(* Logix 5000 project; controller StartingFile_Isaiah_Regacho vendor 1 type 14 code 106 rev 28.11; software revision 28.03 *)

TASK Fault_Logging (periodic, rate 100 ms, priority 10, watchdog 500 ms) : Fault_Logging_Program   // Logs data on faults
TASK MainTask (continuous, watchdog 500 ms) : MainProgram

MODULES
   Local : vendor 1 type 14 code 106 (Compact 0, rev 28.11)
       : 1769-IQ16 (Compact 3, rev 1.1, Input RPI 20 ms)
       : vendor 1 type 7 code 77 (Compact 2, rev 3.1, Input RPI 20 ms)
       : vendor 1 type 7 code 72 (Compact 4, rev 2.1, Output RPI 20 ms)
       : vendor 1 type 7 code 72 (Compact 5, rev 2.1, Output RPI 20 ms)
END_MODULES

TYPE DATE_TIME :
STRUCT
   dateTime : DINT[7];
END_STRUCT
END_TYPE

TYPE FAULTS :
STRUCT
   faultCode : DINT;   // custom fault code depending on type of fault
   timeFaulted : DINT[7];   // time the fault occured
   faultType : DINT;   // minor (1) or major (2) fault
   systemState : DINT;   // current elevator floor state when the fault occured
END_STRUCT
END_TYPE

TYPE LOG_DATA :
STRUCT
   numCalls : DINT;   // keeps track of the # of calls a floor made. also is used for indexing the serviceLog
   timeAve : DINT;   // the average time it takes to service floor
   serviceLog : DATE_TIME[50];   // log of all times a floor was serviced
   timeAcc : DINT;   // keeps track of the TOTAL service time. must divide by numCalls to find average
   timeService : DINT;   // the time it takes to service a floor one instance
END_STRUCT
END_TYPE

ADD_ON_INSTRUCTION getFloorData   (* revision 1.0, ExecutePrescan, ExecuteEnableInFalse *)
// gets floor data and stores in masterLog
VAR_IN_OUT
   floorLogData : LOG_DATA; {required}
END_VAR
VAR
   timeCount : TIMER; {access None}
   logIndex : DINT; {access None}
   false_ons : BOOL; {access None}
END_VAR

ROUTINE EnableInFalse   (* ladder *)
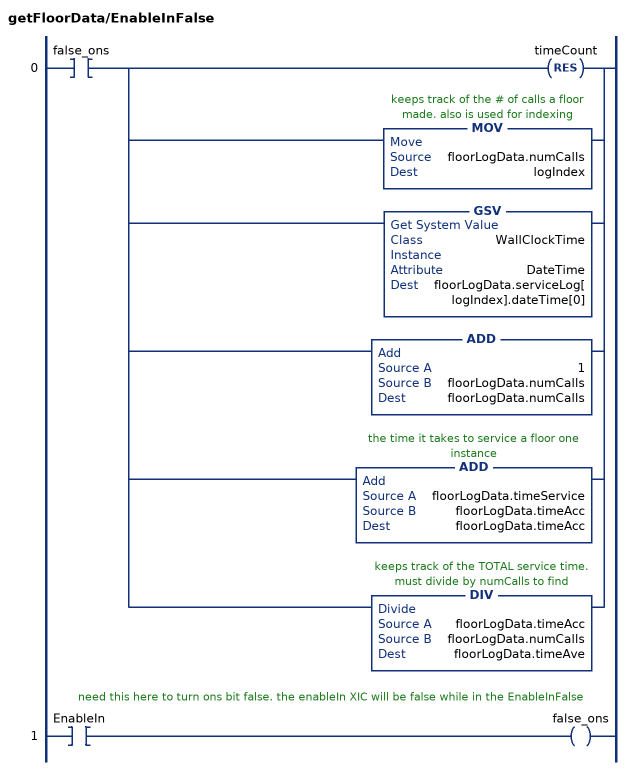
   0: XIC(false_ons)[RES(timeCount) ,MOV(floorLogData.numCalls,logIndex) ,GSV(WallClockTime,,DateTime,floorLogData.serviceLog[logIndex].dateTime[0]) ,ADD(1,floorLogData.numCalls,floorLogData.numCalls) ,ADD(floorLogData.timeService,floorLogData.timeAcc,floorLogData.timeAcc) ,DIV(floorLogData.timeAcc,floorLogData.numCalls,floorLogData.timeAve) ];
   // need this here to turn ons bit false. the enableIn XIC will be false while in the EnableInFalse
   1: XIC(EnableIn)OTE(false_ons);
END_ROUTINE

ROUTINE Logic   (* ladder *)
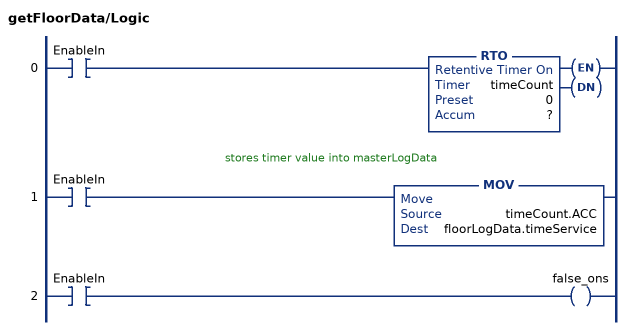
   0: XIC(EnableIn)RTO(timeCount,?,?);
   // stores timer value into masterLogData
   1: XIC(EnableIn)MOV(timeCount.ACC,floorLogData.timeService);
   2: XIC(EnableIn)OTE(false_ons);
END_ROUTINE

ROUTINE Prescan   (* ladder *)
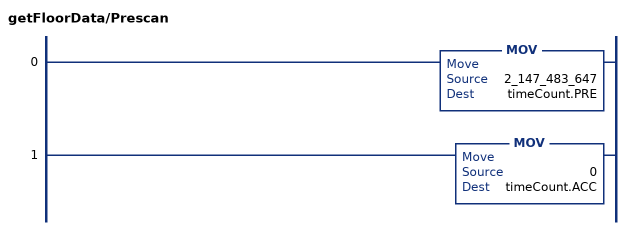
   0: MOV(2_147_483_647,timeCount.PRE);
   1: MOV(0,timeCount.ACC);
END_ROUTINE
END_ADD_ON_INSTRUCTION

PROGRAM Fault_Logging_Program   (* main routine Fault_Logging_Routine *)
VAR
   doorOpenFault_ons : BOOL;
   doorOpenFaultBit : BOOL;
   index : DINT;
   masterFaultLog : FAULTS[10];
   motorRunFault_ons : BOOL;
   motorRunFaultBit : BOOL;
   sensorFault_ons : BOOL;
   sensorFaultBit : BOOL;
END_VAR

ROUTINE Fault_Logging_Routine   (* ladder *)
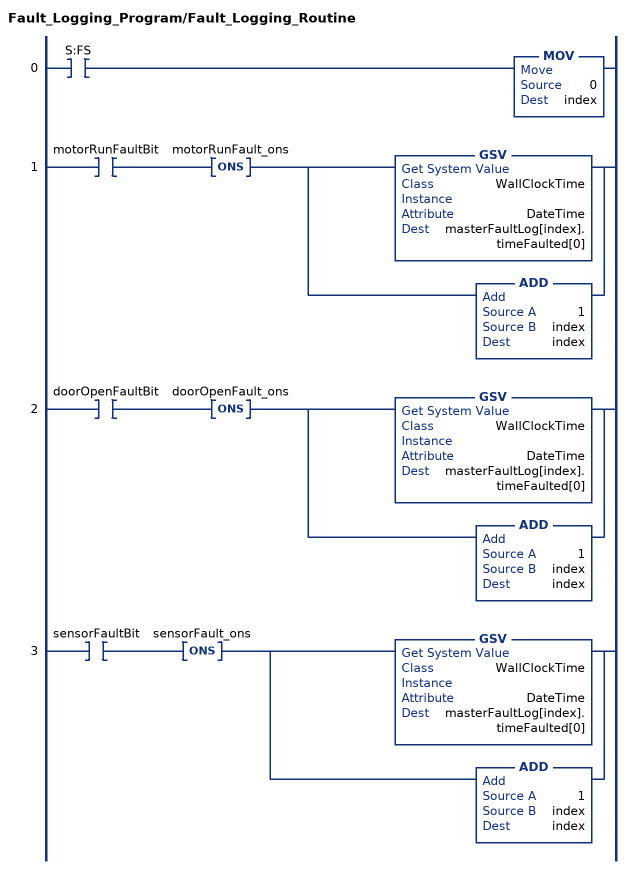
   0: XIC(S:FS)MOV(0,index);
   1: XIC(motorRunFaultBit)ONS(motorRunFault_ons)[GSV(WallClockTime,,DateTime,masterFaultLog[index].timeFaulted[0]) ,ADD(1,index,index) ];
   2: XIC(doorOpenFaultBit)ONS(doorOpenFault_ons)[GSV(WallClockTime,,DateTime,masterFaultLog[index].timeFaulted[0]) ,ADD(1,index,index) ];
   3: XIC(sensorFaultBit)ONS(sensorFault_ons)[GSV(WallClockTime,,DateTime,masterFaultLog[index].timeFaulted[0]) ,ADD(1,index,index) ];
END_ROUTINE
END_PROGRAM

PROGRAM MainProgram   (* main routine MainRoutine *)
VAR
   breakpoint_ons : BOOL;
   callArray : DINT[6] := ([1] := 1, [2] := 2, [4] := 4);
   checkedBothDir : DINT;
   clearFaultsBit : BOOL;
   control_1 : CONTROL := (LEN := 4, EN := 1, IN := 1, FD := 1);
   countDown_ons : BOOL;
   countUp_ons : BOOL;
   CR0 : ALIAS FOR Local:5:O.Data.4;   // Control Relay 0
   Current_State : DINT := 100;
   Current_State_Door : DINT := 1;
   currentFloor : DINT := 4;
   DCLS : ALIAS FOR Local:3:I.Data.8;   // Door Close Limit Switch
   DOLS : ALIAS FOR Local:3:I.Data.9;   // Door Open Limit Switch
   doorOpenFault : TIMER := (PRE := 10000);
   doorOpenFault_ons : BOOL;
   doorOpenFaultBit : BOOL;
   doorOpenFunc : DINT;
   down_ons : BOOL;
   elevatorDirection : DINT;
   faultIndex : DINT;
   FIL1 : ALIAS FOR Local:4:O.Data.11;   // Floor Indicator Light 1
   FIL2 : ALIAS FOR Local:4:O.Data.10;   // Floor Indicator Light 2
   FIL3 : ALIAS FOR Local:4:O.Data.9;   // Floor Indicator Light 3
   FIL4 : ALIAS FOR Local:4:O.Data.8;   // Floor Indicator Light 4
   floor1 : DINT;
   floor1_ons : BOOL;
   floor1Data : getFloorData;
   floor2 : DINT := 1;
   floor2_ons : BOOL;
   floor2Data : getFloorData;
   floor3 : DINT := 2;
   floor3_ons : BOOL;
   floor3Data : getFloorData;
   floor4 : DINT := 3;
   floor4_ons : BOOL;
   floor4Data : getFloorData;
   FLS1 : ALIAS FOR Local:3:I.Data.0;   // Floor Limit Switch 1
   FLS2 : ALIAS FOR Local:3:I.Data.1;   // Floor Limit Switch 2
   FLS3 : ALIAS FOR Local:3:I.Data.2;   // Floor Limit Switch 3
   FLS4 : ALIAS FOR Local:3:I.Data.3;   // Floor Limit Switch 4
   FPB1 : ALIAS FOR Local:2:I.Data.11;   // Floor Pushbutton 1
   FPB2 : ALIAS FOR Local:2:I.Data.10;   // Floor Pushbutton 2
   FPB3 : ALIAS FOR Local:2:I.Data.9;   // Floor Pushbutton 3
   FPB4 : ALIAS FOR Local:2:I.Data.8;   // Floor Pushbutton 4
   IL1 : ALIAS FOR Local:4:O.Data.3;   // Indicator Light 1
   IL2 : ALIAS FOR Local:4:O.Data.2;   // Indicator Light 2
   IL3 : ALIAS FOR Local:4:O.Data.1;   // Indicator Light 3
   IL4 : ALIAS FOR Local:4:O.Data.0;   // Indicator Light 4
   ILC : ALIAS FOR Local:4:O.Data.5;   // Indicator Light Close
   ILE5 : ALIAS FOR Local:4:O.Data.6;   // Indicator Light Emergency 5
   ILO : ALIAS FOR Local:4:O.Data.4;   // Indicator Light Open
   ILTS0 : ALIAS FOR Local:4:O.Data.14;   // Indicator Light Toggle Switch 0
   ILTS1 : ALIAS FOR Local:4:O.Data.13;   // Indicator Light Toggle Switch 1
   ILTS2 : ALIAS FOR Local:4:O.Data.12;   // Indicator Light Toggle Switch 2
   index : DINT := 5;
   logIndex : DINT;
   M0 : ALIAS FOR Local:5:O.Data.0;   // Motor 0
   majorFault_var : DINT := 1;
   masterFaultLog : FAULTS[10];
   masterFaultLog_init : FAULTS[10];
   masterLogData : LOG_DATA[4] := ([0].numCalls := 3, [0].timeAve := 6729, [0].serviceLog[0].dateTime[0] := 2024, [0].serviceLog[0].dateTime[1] := 4, [0].serviceLog[0].dateTime[2] := 11, [0].serviceLog[0].dateTime[3] := 12, [0].serviceLog[0].dateTime[4] := 6, [0].serviceLog[0].dateTime[5] := 16, [0].serviceLog[0].dateTime[6] := 127621, [0].serviceLog[1].dateTime[0] := 2024, [0].serviceLog[1].dateTime[1] := 4, [0].serviceLog[1].dateTime[2] := 11, [0].serviceLog[1].dateTime[3] := 12, [0].serviceLog[1].dateTime[4] := 6, [0].serviceLog[1].dateTime[5] := 34, [0].serviceLog[1].dateTime[6] := 745369, [0].serviceLog[2].dateTime[0] := 2024, [0].serviceLog[2].dateTime[1] := 4, [0].serviceLog[2].dateTime[2] := 11, [0].serviceLog[2].dateTime[3] := 12, [0].serviceLog[2].dateTime[4] := 7, [0].serviceLog[2].dateTime[5] := 4, [0].serviceLog[2].dateTime[6] := 869689, [0].timeAcc := 20188, [0].timeService := 363313, [1].numCalls := 2, [1].timeAve := 12433, [1].serviceLog[0].dateTime[0] := 2024, [1].serviceLog[0].dateTime[1] := 4, [1].serviceLog[0].dateTime[2] := 11, [1].serviceLog[0].dateTime[3] := 12, [1].serviceLog[0].dateTime[4] := 6, [1].serviceLog[0].dateTime[5] := 10, [1].serviceLog[0].dateTime[6] := 288799, [1].serviceLog[1].dateTime[0] := 2024, [1].serviceLog[1].dateTime[1] := 4, [1].serviceLog[1].dateTime[2] := 11, [1].serviceLog[1].dateTime[3] := 12, [1].serviceLog[1].dateTime[4] := 6, [1].serviceLog[1].dateTime[5] := 45, [1].serviceLog[1].dateTime[6] := 652417, [1].timeAcc := 24866, [1].timeService := 363928, [3].numCalls := 4, [3].timeAve := 8386, [3].serviceLog[0].dateTime[0] := 2024, [3].serviceLog[0].dateTime[1] := 4, [3].serviceLog[0].dateTime[2] := 11, [3].serviceLog[0].dateTime[3] := 12, [3].serviceLog[0].dateTime[4] := 6, [3].serviceLog[0].dateTime[5] := 3, [3].serviceLog[0].dateTime[6] := 427814, [3].serviceLog[1].dateTime[0] := 2024, [3].serviceLog[1].dateTime[1] := 4, [3].serviceLog[1].dateTime[2] := 11, [3].serviceLog[1].dateTime[3] := 12, [3].serviceLog[1].dateTime[4] := 6, [3].serviceLog[1].dateTime[5] := 22, [3].serviceLog[1].dateTime[6] := 780797, [3].serviceLog[2].dateTime[0] := 2024,
        [3].serviceLog[2].dateTime[1] := 4, [3].serviceLog[2].dateTime[2] := 11, [3].serviceLog[2].dateTime[3] := 12, [3].serviceLog[2].dateTime[4] := 6, [3].serviceLog[2].dateTime[5] := 49, [3].serviceLog[2].dateTime[6] := 470088, [3].serviceLog[3].dateTime[0] := 2024, [3].serviceLog[3].dateTime[1] := 4, [3].serviceLog[3].dateTime[2] := 11, [3].serviceLog[3].dateTime[3] := 12, [3].serviceLog[3].dateTime[4] := 6, [3].serviceLog[3].dateTime[5] := 56, [3].serviceLog[3].dateTime[6] := 856063, [3].timeAcc := 33544, [3].timeService := 364724);
   masterLogData_init : LOG_DATA[4];
   motorRunFault : TIMER := (PRE := 8000);
   motorRunFault_ons : BOOL;
   motorRunFaultBit : BOOL;
   Next_State : DINT := 100;
   Next_State_Door : DINT := 1;
   nextFloor : DINT := 4;
   PB1 : ALIAS FOR Local:2:I.Data.3;   // Pushbutton 1
   PB2 : ALIAS FOR Local:2:I.Data.2;   // Pushbutton 2
   PB3 : ALIAS FOR Local:2:I.Data.1;   // Pushbutton 3
   PB4 : ALIAS FOR Local:2:I.Data.0;   // Pushbutton 4
   PBC : ALIAS FOR Local:2:I.Data.5;   // Pushbutton Close
   PBE5 : ALIAS FOR Local:2:I.Data.6;   // Pushbutton Emergency 5
   PBO : ALIAS FOR Local:2:I.Data.4;   // Pushbutton Open
   sensorFault_ons : BOOL;
   sensorFaultBit : BOOL;
   SOL0 : ALIAS FOR Local:5:O.Data.2;   // Solenoid 0
   START : ALIAS FOR Local:2:I.Data.14;   // Start Button (N.O.)
   STOP : ALIAS FOR Local:2:I.Data.15;   // Stop Button (N.C.)
   test2_ons : BOOL;
   test_ons : BOOL;
   timer3sec : TIMER := (PRE := 3000, ACC := 3000, EN := 1, DN := 1);
   timer3secVar : DINT := 1;
   timer5sec : TIMER := (PRE := 5000, ACC := 5000, EN := 1, DN := 1);
   TS0 : ALIAS FOR Local:3:I.Data.12;   // Toggle Switch 0
   TS1 : ALIAS FOR Local:3:I.Data.11;   // Toggle Switch 1
   TS2 : ALIAS FOR Local:3:I.Data.10;   // Toggle Switch 2
   up_ons : BOOL;
   V_CR0 : BOOL;   // Virtual Control Relay 0
   V_DCLS : BOOL;   // Virtual Door Close Limit Switch
   V_DOLS : BOOL := 1;   // Virtual Door Open Limit Switch
   V_FIL1 : BOOL := 1;   // Virtual Floor Indicator Light 1
   V_FIL2 : BOOL := 1;   // Virtual Floor Indicator Light 2
   V_FIL3 : BOOL;   // Virtual Floor Indicator Light 3
   V_FIL4 : BOOL := 1;   // Virtual Floor Indicator Light 4
   V_FLS1 : BOOL;   // Virtual Floor Limit Switch 1
   V_FLS2 : BOOL;   // Virtual Floor Limit Switch 2
   V_FLS3 : BOOL;   // Virtual Floor Limit Switch 3
   V_FLS4 : BOOL;   // Virtual Floor Limit Switch 4
   V_FPB1 : BOOL;   // Virtual Floor Pushbutton 1
   V_FPB2 : BOOL;   // Virtual Floor Pushbutton 2
   V_FPB3 : BOOL;   // Virtual Floor Pushbutton 3
   V_FPB4 : BOOL;   // Virtual Floor Pushbutton 4
   V_IL1 : BOOL := 1;   // Virtual Indicator Light 1
   V_IL2 : BOOL := 1;   // Virtual Indicator Light 2
   V_IL3 : BOOL;   // Virtual Indicator Light 3
   V_IL4 : BOOL := 1;   // Virtual Indicator Light 4
   V_ILC : BOOL := 1;   // Virtual Indicator Light Close
   V_ILE5 : BOOL := 1;   // Virtual Indicator Light Emergency 5
   V_ILO : BOOL;   // Virtual Indicator Light Open
   V_ILTS0 : BOOL;   // Vitual Indicator Light Toggle Switch 0
   V_ILTS1 : BOOL;   // Virtual Indicator Light Toggle Switch 1
   V_ILTS2 : BOOL;   // Virtual Indicator Light Toggle Switch 2
   V_M0 : BOOL;   // Virtual Motor 0
   V_PB1 : BOOL;   // Virtual Pushbutton 1
   V_PB2 : BOOL;   // Virtual Pushbutton 2
   V_PB3 : BOOL;   // Virtual Pushbutton 3
   V_PB4 : BOOL;   // Virtual Pushbutton 4
   V_PBC : BOOL;   // Virtual Pushbutton Close
   V_PBE5 : BOOL;   // Virtual Pushbutton Emergency 5
   V_PBO : BOOL;   // Virtual Pushbutton Open
   V_SOL0 : BOOL := 1;   // Virtual Solenoid 0
   V_START : BOOL;   // Virtual Start Button (N.O.)
   V_STOP : BOOL := 1;   // Virtual Stop Button (N.C.)
   V_TS0 : BOOL := 1;   // Virtual Toggle Switch 0
   V_TS1 : BOOL;   // Virtual Toggle Switch 1
   V_TS2 : BOOL;   // Virtual Toggle Switch 2
END_VAR

ROUTINE BufferInput   (* ladder *)
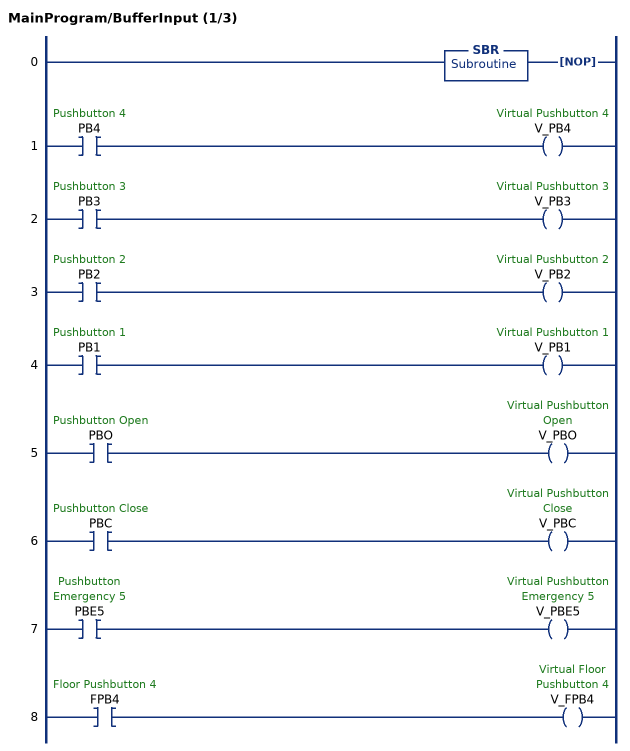
   0: SBR()NOP();
   1: XIC(PB4)OTE(V_PB4);
   2: XIC(PB3)OTE(V_PB3);
   3: XIC(PB2)OTE(V_PB2);
   4: XIC(PB1)OTE(V_PB1);
   5: XIC(PBO)OTE(V_PBO);
   6: XIC(PBC)OTE(V_PBC);
   7: XIC(PBE5)OTE(V_PBE5);
   8: XIC(FPB4)OTE(V_FPB4);
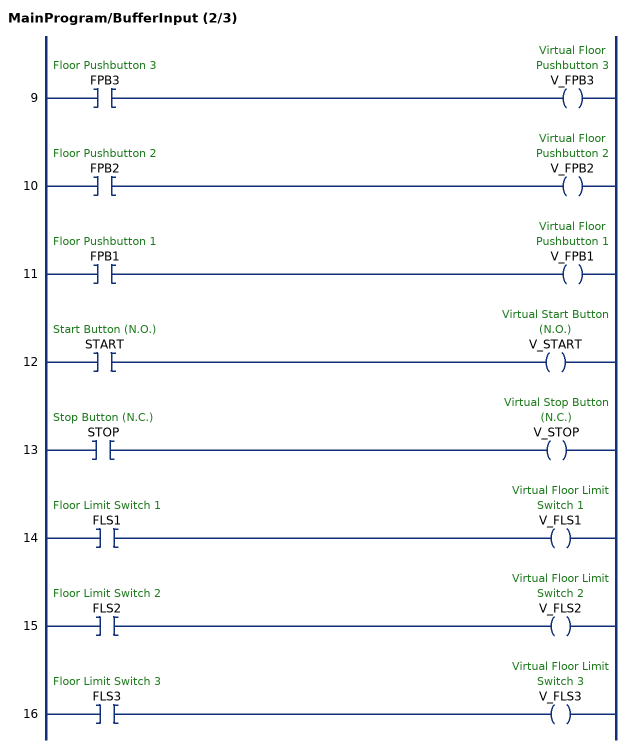
   9: XIC(FPB3)OTE(V_FPB3);
   10: XIC(FPB2)OTE(V_FPB2);
   11: XIC(FPB1)OTE(V_FPB1);
   12: XIC(START)OTE(V_START);
   13: XIC(STOP)OTE(V_STOP);
   14: XIC(FLS1)OTE(V_FLS1);
   15: XIC(FLS2)OTE(V_FLS2);
   16: XIC(FLS3)OTE(V_FLS3);
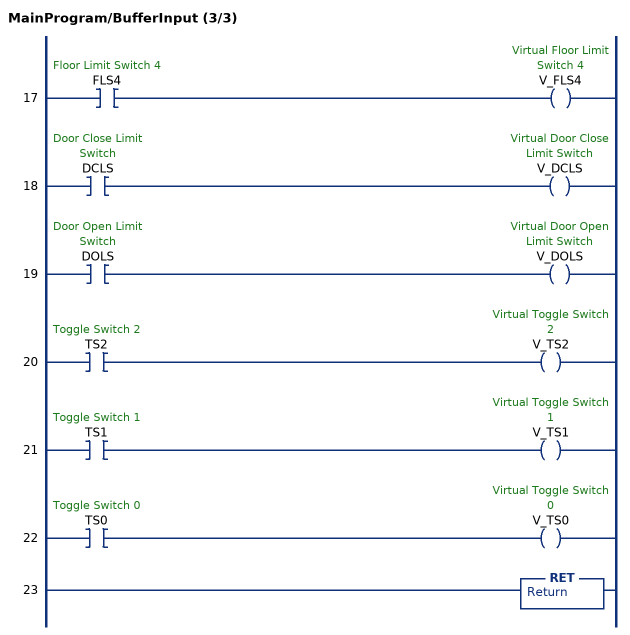
   17: XIC(FLS4)OTE(V_FLS4);
   18: XIC(DCLS)OTE(V_DCLS);
   19: XIC(DOLS)OTE(V_DOLS);
   20: XIC(TS2)OTE(V_TS2);
   21: XIC(TS1)OTE(V_TS1);
   22: XIC(TS0)OTE(V_TS0);
   23: RET();
END_ROUTINE

ROUTINE BufferOutput   (* ladder *)
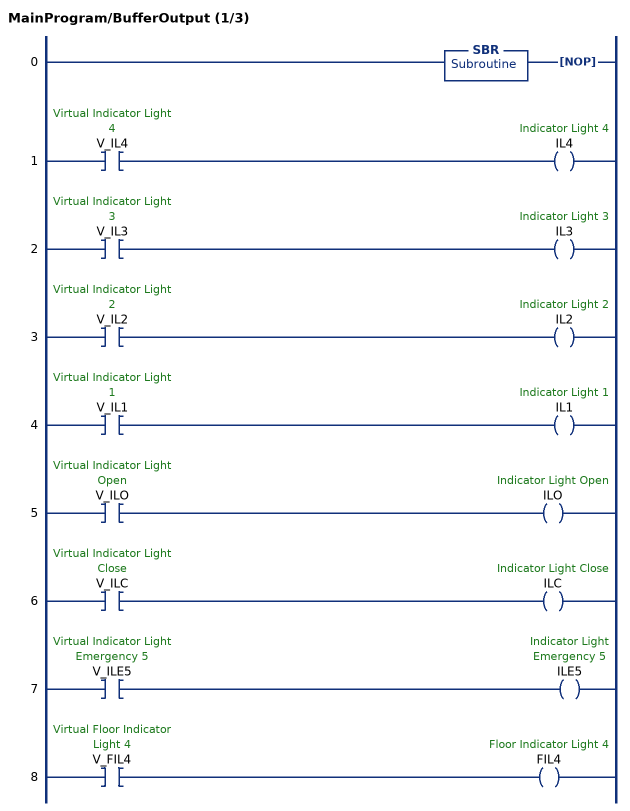
   0: SBR()NOP();
   1: XIC(V_IL4)OTE(IL4);
   2: XIC(V_IL3)OTE(IL3);
   3: XIC(V_IL2)OTE(IL2);
   4: XIC(V_IL1)OTE(IL1);
   5: XIC(V_ILO)OTE(ILO);
   6: XIC(V_ILC)OTE(ILC);
   7: XIC(V_ILE5)OTE(ILE5);
   8: XIC(V_FIL4)OTE(FIL4);
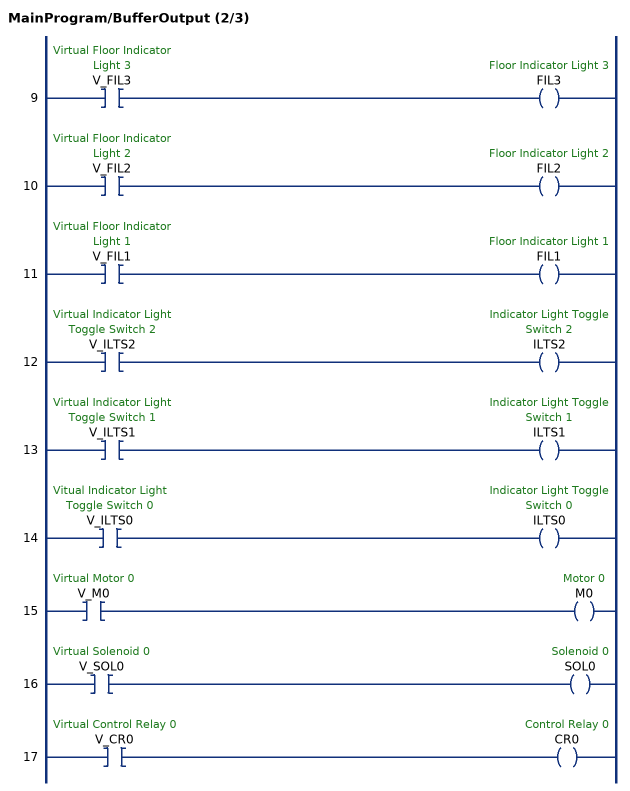
   9: XIC(V_FIL3)OTE(FIL3);
   10: XIC(V_FIL2)OTE(FIL2);
   11: XIC(V_FIL1)OTE(FIL1);
   12: XIC(V_ILTS2)OTE(ILTS2);
   13: XIC(V_ILTS1)OTE(ILTS1);
   14: XIC(V_ILTS0)OTE(ILTS0);
   15: XIC(V_M0)OTE(M0);
   16: XIC(V_SOL0)OTE(SOL0);
   17: XIC(V_CR0)OTE(CR0);
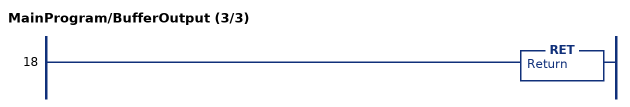
   18: RET();
END_ROUTINE

ROUTINE Door_State_Machine   (* ladder *)
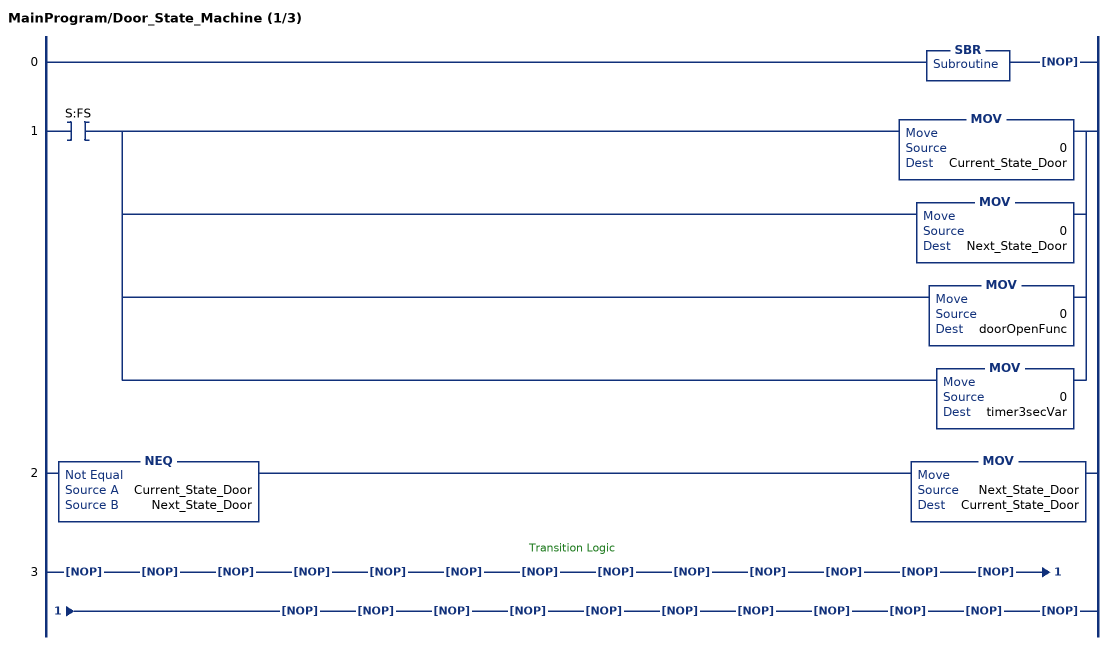
   0: SBR()NOP();
   1: XIC(S:FS)[MOV(0,Current_State_Door) ,MOV(0,Next_State_Door) ,MOV(0,doorOpenFunc) ,MOV(0,timer3secVar) ];
   2: NEQ(Current_State_Door,Next_State_Door)MOV(Next_State_Door,Current_State_Door);
   // Transition Logic
   3: NOP()NOP()NOP()NOP()NOP()NOP()NOP()NOP()NOP()NOP()NOP()NOP()NOP()NOP()NOP()NOP()NOP()NOP()NOP()NOP()NOP()NOP()NOP()NOP();
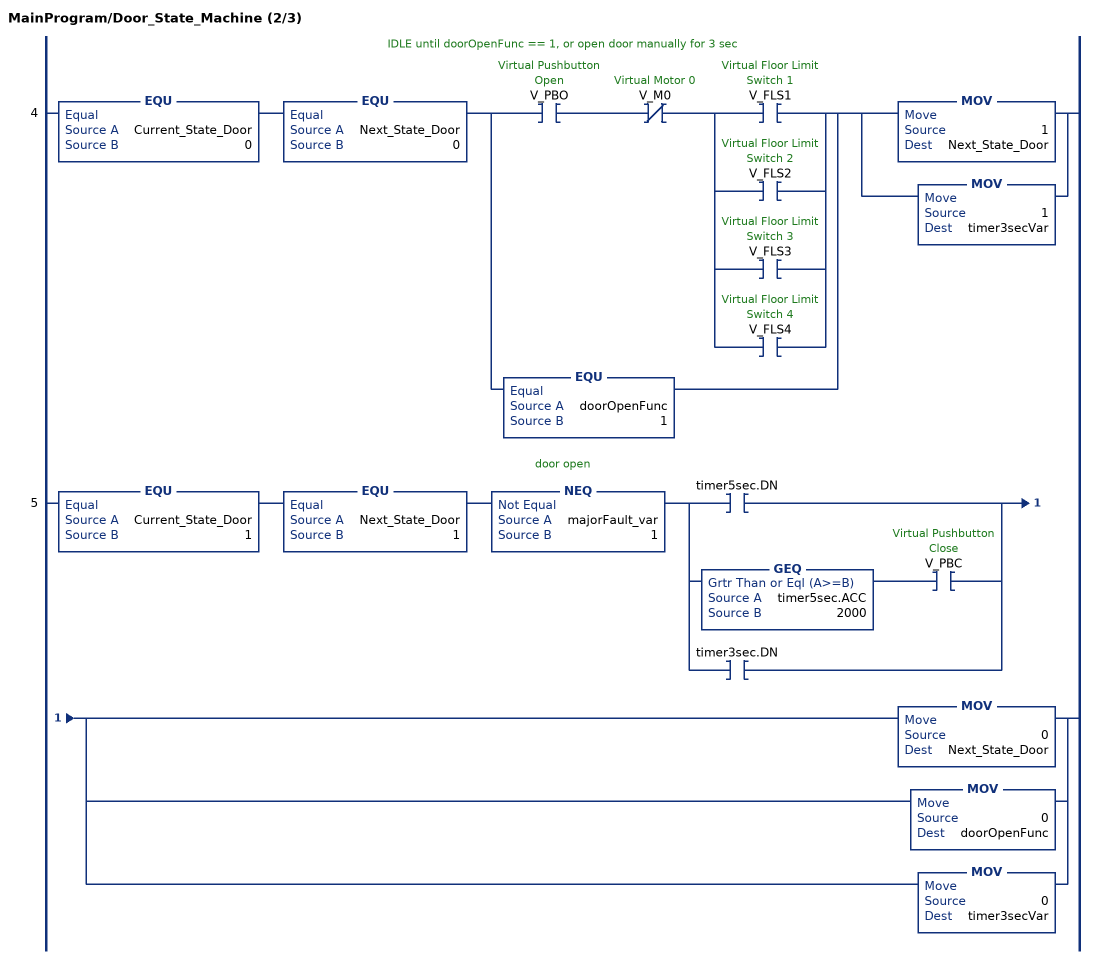
   // IDLE until doorOpenFunc == 1, or open door manually for 3 sec
   4: EQU(Current_State_Door,0)EQU(Next_State_Door,0)[XIC(V_PBO) XIO(V_M0) [XIC(V_FLS1) ,XIC(V_FLS2) ,XIC(V_FLS3) ,XIC(V_FLS4) ] ,EQU(doorOpenFunc,1) ][MOV(1,Next_State_Door) ,MOV(1,timer3secVar) ];
   // door open
   5: EQU(Current_State_Door,1)EQU(Next_State_Door,1)NEQ(majorFault_var,1)[XIC(timer5sec.DN) ,GEQ(timer5sec.ACC,2000) XIC(V_PBC) ,XIC(timer3sec.DN) ][MOV(0,Next_State_Door) ,MOV(0,doorOpenFunc) ,MOV(0,timer3secVar) ];
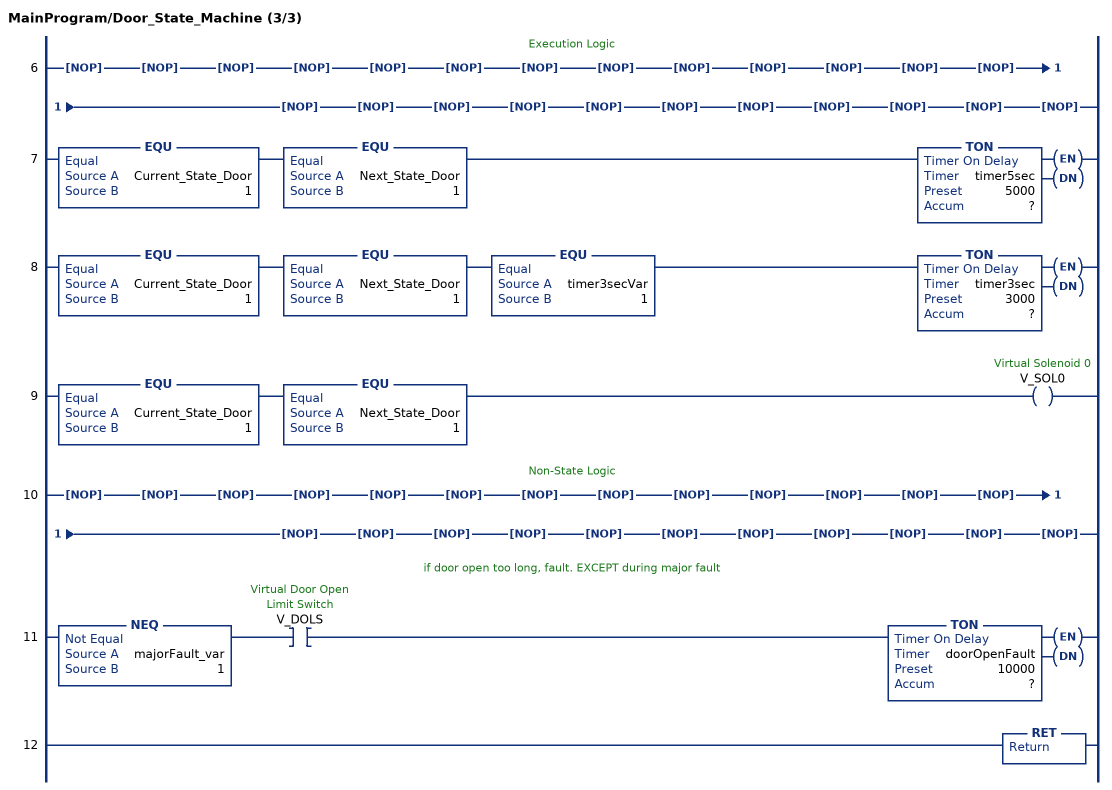
   // Execution Logic
   6: NOP()NOP()NOP()NOP()NOP()NOP()NOP()NOP()NOP()NOP()NOP()NOP()NOP()NOP()NOP()NOP()NOP()NOP()NOP()NOP()NOP()NOP()NOP()NOP();
   7: EQU(Current_State_Door,1)EQU(Next_State_Door,1)TON(timer5sec,?,?);
   8: EQU(Current_State_Door,1)EQU(Next_State_Door,1)EQU(timer3secVar,1)TON(timer3sec,?,?);
   9: EQU(Current_State_Door,1)EQU(Next_State_Door,1)OTE(V_SOL0);
   // Non-State Logic
   10: NOP()NOP()NOP()NOP()NOP()NOP()NOP()NOP()NOP()NOP()NOP()NOP()NOP()NOP()NOP()NOP()NOP()NOP()NOP()NOP()NOP()NOP()NOP()NOP();
   // if door open too long, fault. EXCEPT during major fault
   11: NEQ(majorFault_var,1)XIC(V_DOLS)TON(doorOpenFault,?,?);
   12: RET();
END_ROUTINE

ROUTINE Floor_State_Machine   (* ladder *)
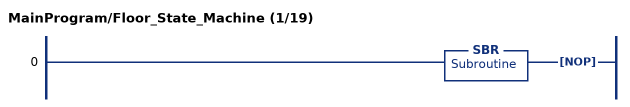
   0: SBR()NOP();
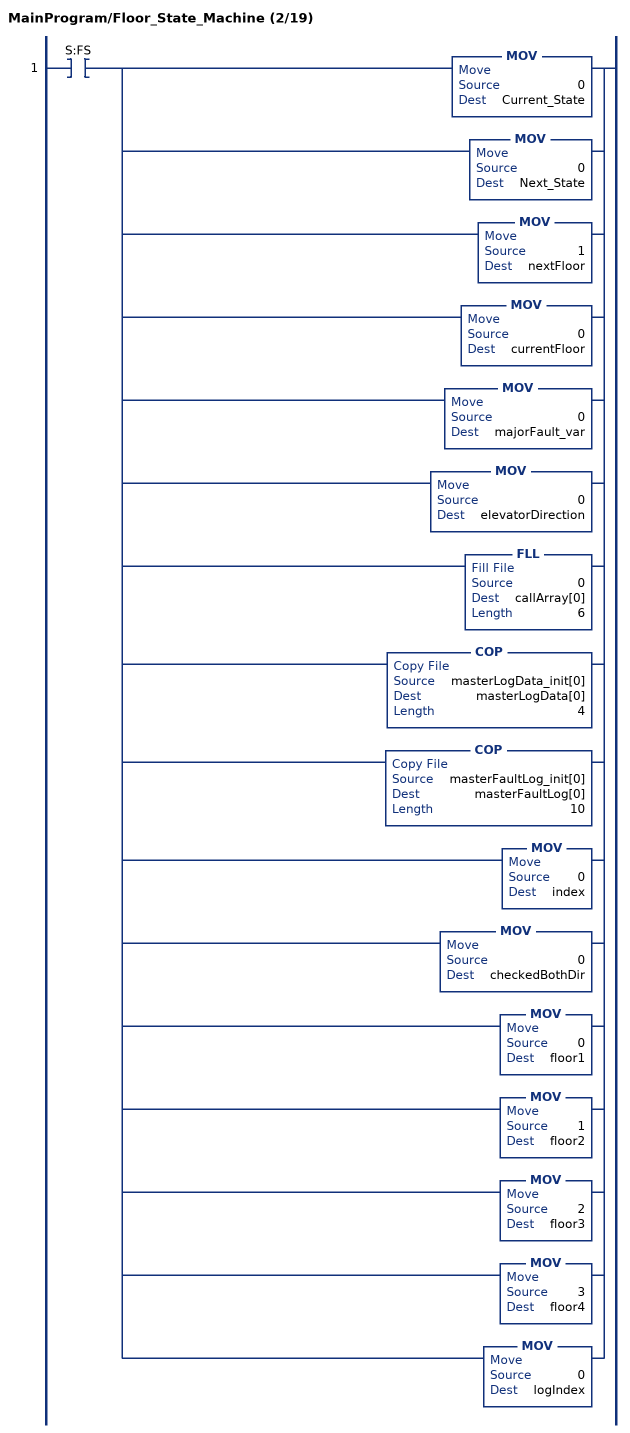
   1: XIC(S:FS)[MOV(0,Current_State) ,MOV(0,Next_State) ,MOV(1,nextFloor) ,MOV(0,currentFloor) ,MOV(0,majorFault_var) ,MOV(0,elevatorDirection) ,FLL(0,callArray[0],6) ,COP(masterLogData_init[0],masterLogData[0],4) ,COP(masterFaultLog_init[0],masterFaultLog[0],10) ,MOV(0,index) ,MOV(0,checkedBothDir) ,MOV(0,floor1) ,MOV(1,floor2) ,MOV(2,floor3) ,MOV(3,floor4) ,MOV(0,logIndex) ];
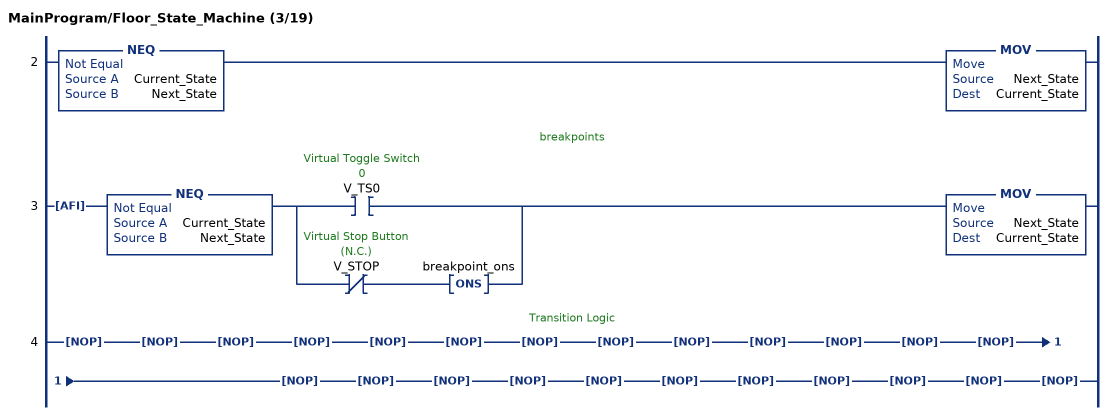
   2: NEQ(Current_State,Next_State)MOV(Next_State,Current_State);
   // breakpoints
   3: AFI()NEQ(Current_State,Next_State)[XIC(V_TS0) ,XIO(V_STOP) ONS(breakpoint_ons) ]MOV(Next_State,Current_State);
   // Transition Logic
   4: NOP()NOP()NOP()NOP()NOP()NOP()NOP()NOP()NOP()NOP()NOP()NOP()NOP()NOP()NOP()NOP()NOP()NOP()NOP()NOP()NOP()NOP()NOP()NOP();
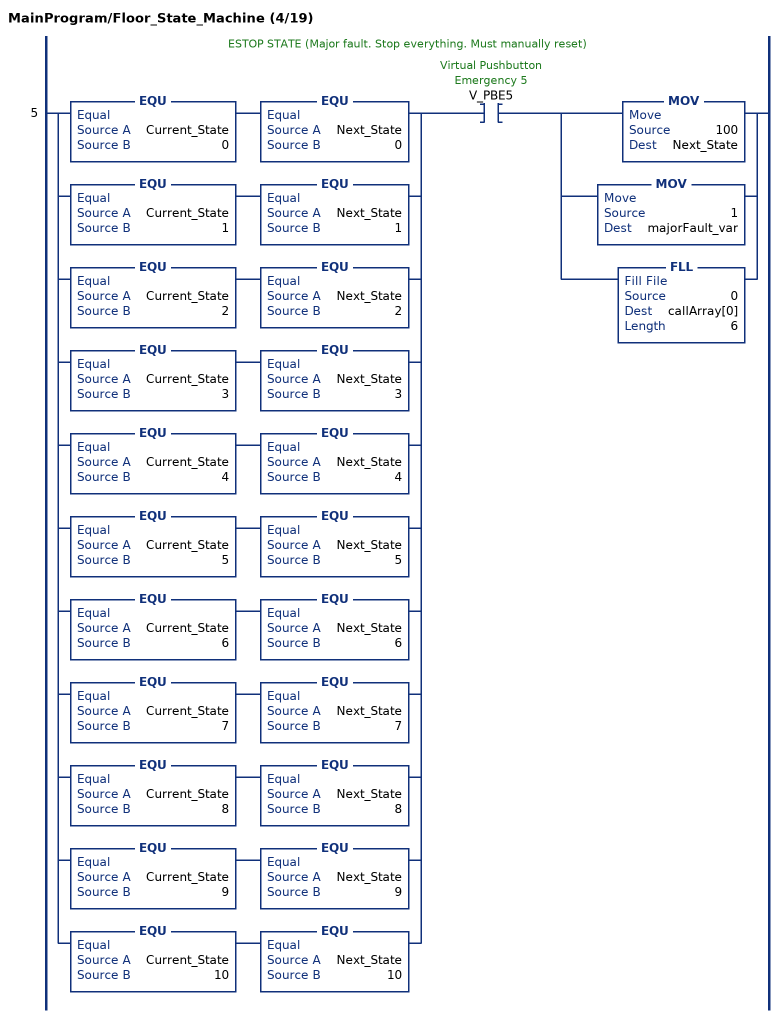
   // ESTOP STATE (Major fault. Stop everything. Must manually reset)
   5: [EQU(Current_State,0) EQU(Next_State,0) ,EQU(Current_State,1) EQU(Next_State,1) ,EQU(Current_State,2) EQU(Next_State,2) ,EQU(Current_State,3) EQU(Next_State,3) ,EQU(Current_State,4) EQU(Next_State,4) ,EQU(Current_State,5) EQU(Next_State,5) ,EQU(Current_State,6) EQU(Next_State,6) ,EQU(Current_State,7) EQU(Next_State,7) ,EQU(Current_State,8) EQU(Next_State,8) ,EQU(Current_State,9) EQU(Next_State,9) ,EQU(Current_State,10) EQU(Next_State,10) ]XIC(V_PBE5)[MOV(100,Next_State) ,MOV(1,majorFault_var) ,FLL(0,callArray[0],6) ];
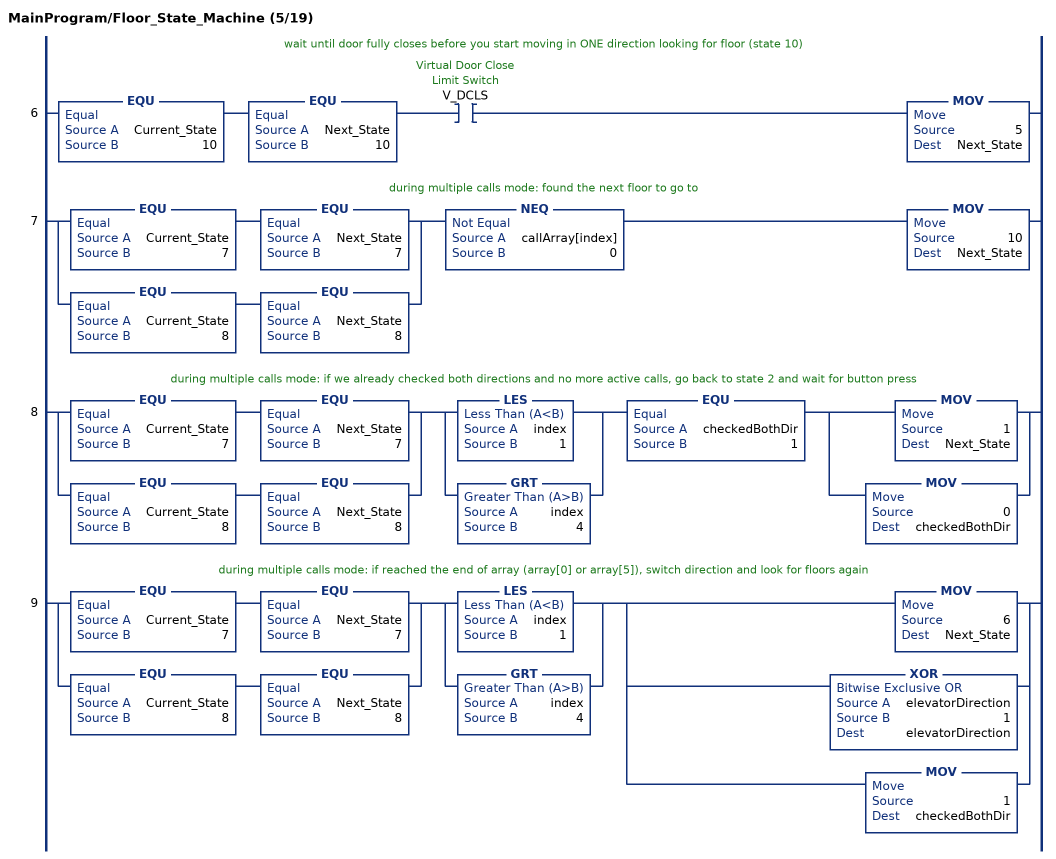
   // wait until door fully closes before you start moving in ONE direction looking for floor (state 10)
   6: EQU(Current_State,10)EQU(Next_State,10)XIC(V_DCLS)MOV(5,Next_State);
   // during multiple calls mode: found the next floor to go to
   7: [EQU(Current_State,7) EQU(Next_State,7) ,EQU(Current_State,8) EQU(Next_State,8) ]NEQ(callArray[index],0)MOV(10,Next_State);
   // during multiple calls mode: if we already checked both directions and no more active calls, go back to state 2 and wait for button press
   8: [EQU(Current_State,7) EQU(Next_State,7) ,EQU(Current_State,8) EQU(Next_State,8) ][LES(index,1) ,GRT(index,4) ]EQU(checkedBothDir,1)[MOV(1,Next_State) ,MOV(0,checkedBothDir) ];
   // during multiple calls mode: if reached the end of array (array[0] or array[5]), switch direction and look for floors again
   9: [EQU(Current_State,7) EQU(Next_State,7) ,EQU(Current_State,8) EQU(Next_State,8) ][LES(index,1) ,GRT(index,4) ][MOV(6,Next_State) ,XOR(elevatorDirection,1,elevatorDirection) ,MOV(1,checkedBothDir) ];
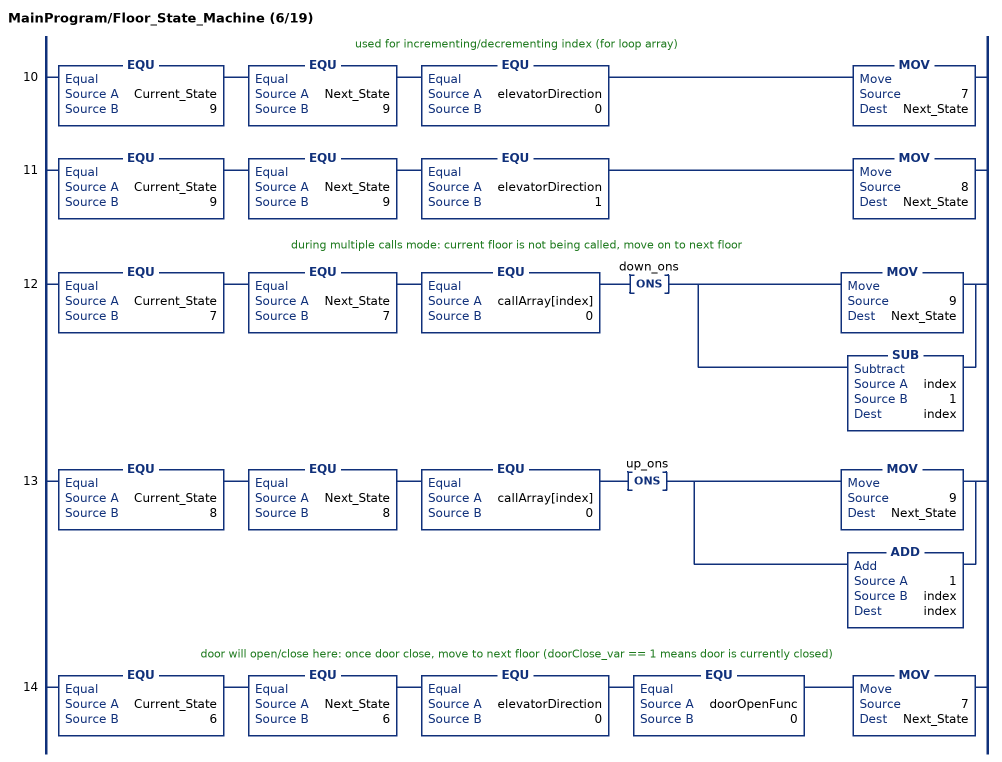
   // used for incrementing/decrementing index (for loop array)
   10: EQU(Current_State,9)EQU(Next_State,9)EQU(elevatorDirection,0)MOV(7,Next_State);
   11: EQU(Current_State,9)EQU(Next_State,9)EQU(elevatorDirection,1)MOV(8,Next_State);
   // during multiple calls mode: current floor is not being called, move on to next floor
   12: EQU(Current_State,7)EQU(Next_State,7)EQU(callArray[index],0)ONS(down_ons)[MOV(9,Next_State) ,SUB(index,1,index) ];
   13: EQU(Current_State,8)EQU(Next_State,8)EQU(callArray[index],0)ONS(up_ons)[MOV(9,Next_State) ,ADD(1,index,index) ];
   // door will open/close here: once door close, move to next floor (doorClose_var == 1 means door is currently closed)
   14: EQU(Current_State,6)EQU(Next_State,6)EQU(elevatorDirection,0)EQU(doorOpenFunc,0)MOV(7,Next_State);
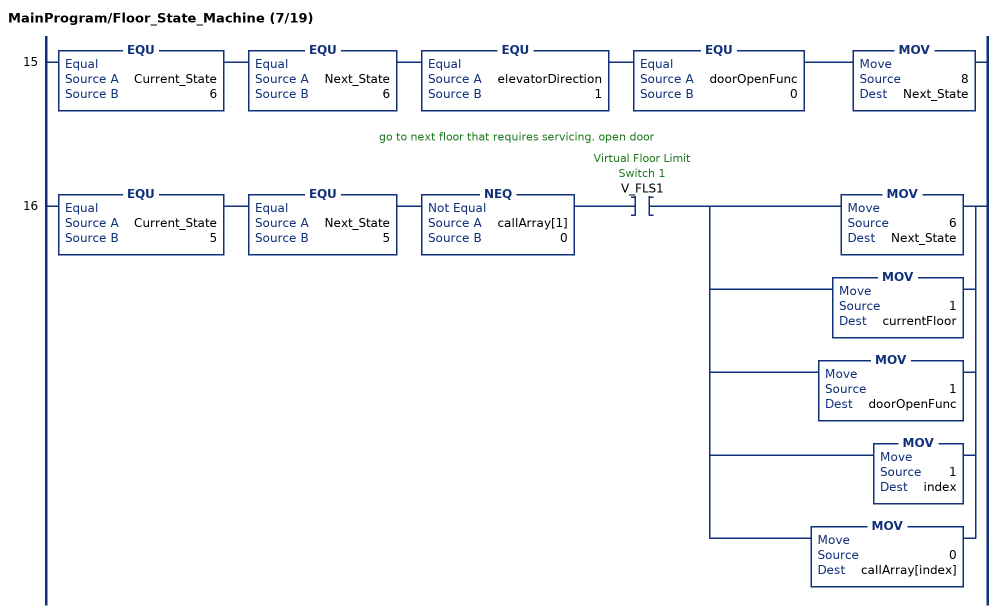
   15: EQU(Current_State,6)EQU(Next_State,6)EQU(elevatorDirection,1)EQU(doorOpenFunc,0)MOV(8,Next_State);
   // go to next floor that requires servicing. open door
   16: EQU(Current_State,5)EQU(Next_State,5)NEQ(callArray[1],0)XIC(V_FLS1)[MOV(6,Next_State) ,MOV(1,currentFloor) ,MOV(1,doorOpenFunc) ,MOV(1,index) ,MOV(0,callArray[index]) ];
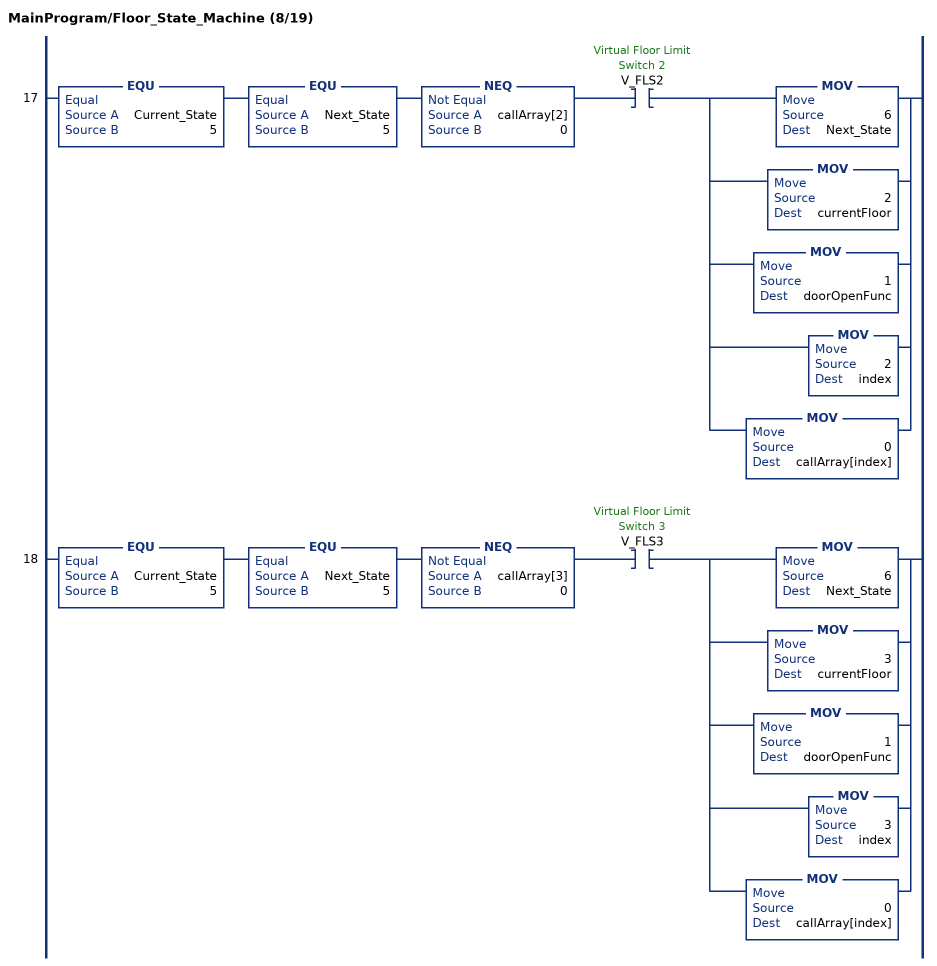
   17: EQU(Current_State,5)EQU(Next_State,5)NEQ(callArray[2],0)XIC(V_FLS2)[MOV(6,Next_State) ,MOV(2,currentFloor) ,MOV(1,doorOpenFunc) ,MOV(2,index) ,MOV(0,callArray[index]) ];
   18: EQU(Current_State,5)EQU(Next_State,5)NEQ(callArray[3],0)XIC(V_FLS3)[MOV(6,Next_State) ,MOV(3,currentFloor) ,MOV(1,doorOpenFunc) ,MOV(3,index) ,MOV(0,callArray[index]) ];
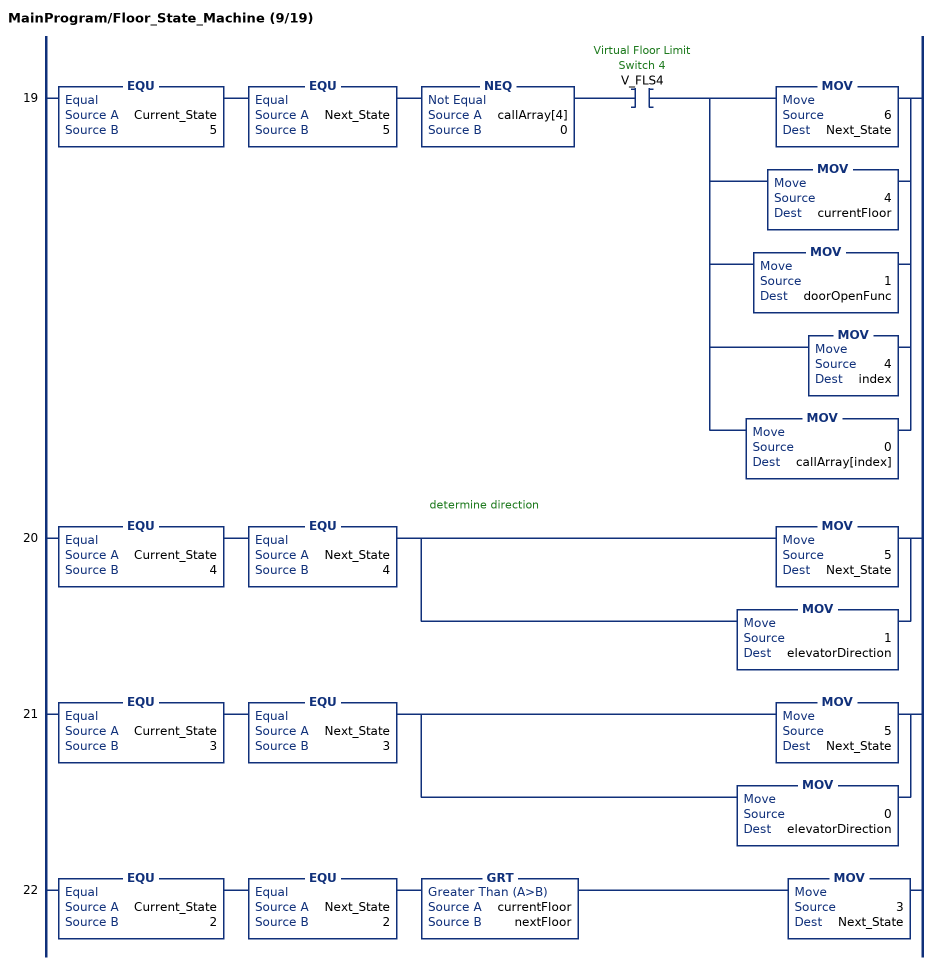
   19: EQU(Current_State,5)EQU(Next_State,5)NEQ(callArray[4],0)XIC(V_FLS4)[MOV(6,Next_State) ,MOV(4,currentFloor) ,MOV(1,doorOpenFunc) ,MOV(4,index) ,MOV(0,callArray[index]) ];
   // determine direction
   20: EQU(Current_State,4)EQU(Next_State,4)[MOV(5,Next_State) ,MOV(1,elevatorDirection) ];
   21: EQU(Current_State,3)EQU(Next_State,3)[MOV(5,Next_State) ,MOV(0,elevatorDirection) ];
   22: EQU(Current_State,2)EQU(Next_State,2)GRT(currentFloor,nextFloor)MOV(3,Next_State);
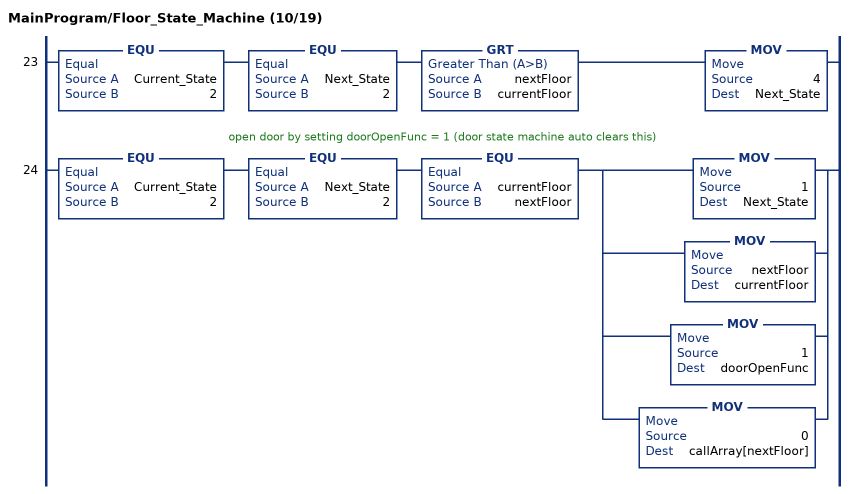
   23: EQU(Current_State,2)EQU(Next_State,2)GRT(nextFloor,currentFloor)MOV(4,Next_State);
   // open door by setting doorOpenFunc = 1 (door state machine auto clears this)
   24: EQU(Current_State,2)EQU(Next_State,2)EQU(currentFloor,nextFloor)[MOV(1,Next_State) ,MOV(nextFloor,currentFloor) ,MOV(1,doorOpenFunc) ,MOV(0,callArray[nextFloor]) ];
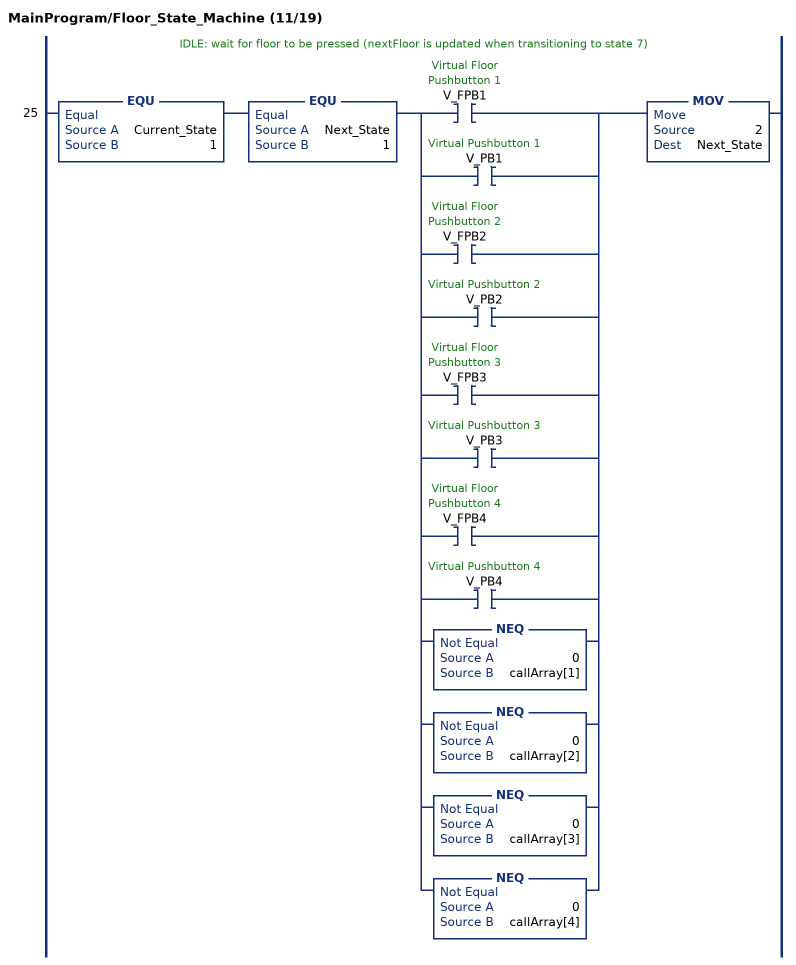
   // IDLE: wait for floor to be pressed (nextFloor is updated when transitioning to state 7)
   25: EQU(Current_State,1)EQU(Next_State,1)[XIC(V_FPB1) ,XIC(V_PB1) ,XIC(V_FPB2) ,XIC(V_PB2) ,XIC(V_FPB3) ,XIC(V_PB3) ,XIC(V_FPB4) ,XIC(V_PB4) ,NEQ(0,callArray[1]) ,NEQ(0,callArray[2]) ,NEQ(0,callArray[3]) ,NEQ(0,callArray[4]) ]MOV(2,Next_State);
